Omron CX-Programmer project NewProject (CX-Programmer 9.75)

# PLC NewPLC1: CP2E-N N

## Global symbols (name address type ; comment)
0.00 BOOL  ; PB Start M1
0.01 BOOL  ; PB Stop M1
0.02 BOOL  ; SS FWD M1
0.03 BOOL  ; SS RVS M1
0.04 BOOL  ; Emergency Stop
0.05 BOOL  ; Sensor M1
0.06 BOOL  ; Trip CNT M1
100.00 BOOL  ; Trip M1
100.01 BOOL  ; Contactor M1
100.02 BOOL  ; Relay FWD M1
100.03 BOOL  ; Relay RVS M1
101.00 BOOL  ; Trip M2
101.01 BOOL  ; Contactor M2
101.02 BOOL  ; Relay FWD M2
101.03 BOOL  ; Relay RVS M2
170.01 BOOL  ; LOCK START FWD VER
1.00 BOOL  ; PB Start M2
1.01 BOOL  ; PB Stop M2
1.02 BOOL  ; SS FWD M2
1.03 BOOL  ; SS RVS M2
1.04 BOOL  ; Sensor M2
1.05 BOOL  ; Trip CNT M2
21.00 BOOL  ; ls vertical fwd
21.01 BOOL  ; ls vertical rev
21.02 BOOL  ; ls horizontal fwd
21.03 BOOL  ; ls horizontal rev
60.00 BOOL  ; M1_achieved'
70.01 BOOL  ; LOCK START FWD HOR
70.02 BOOL  ; LOCK START REV HOR
C000 BOOL  ; Siklus M1
C001 BOOL  ; Siklus M2
C002 BOOL  ; Siklus M1
C003 BOOL  ; Siklus M2
C010 BOOL  ; Siklus (1) M1
C011 BOOL  ; Siklus (2) M1
C110 BOOL  ; Siklus (1) M2
C111 BOOL  ; Siklus (2) M2
D0 CHANNEL  ; Input Siklus M1
D10 CHANNEL  ; Input Siklus M2
D100 CHANNEL  ; '
D20 CHANNEL  ; Input Siklus M1
D30 CHANNEL  ; Input Siklus M2
D5400 CHANNEL  ; Counter_test
D5410 CHANNEL  ; Counter_target
D600 CHANNEL  ; Input Siklus M1
D660 CHANNEL  ; Input Siklus M2
W0.00 BOOL  ; H.PB Start M1
W0.01 BOOL  ; H.PB Stop M1
W0.02 BOOL  ; H.SS FWD M1
W0.03 BOOL  ; H.SS RVS M1
W0.04 BOOL  ; H.Emergency Stop
W0.05 BOOL  ; H.Sensor M1
W0.06 BOOL  ; H.Trip CNT M1
W0.07 BOOL  ; LS Left M1
W0.08 BOOL  ; LS Right M1
W100.00 BOOL  ; H.Trip M1
W100.01 BOOL  ; H.CONTACTOR M1
W100.02 BOOL  ; H.Relay FWD M1
W100.03 BOOL  ; H.Relay RVS M1
W101.00 BOOL  ; H.Trip M2
W101.01 BOOL  ; H.CONTACTOR M2
W101.02 BOOL  ; H.Relay FWD M2
W101.03 BOOL  ; H.Relay RVS M2
W1.00 BOOL  ; H.PB Start M2
W1.01 BOOL  ; H.PB Stop M2
W1.02 BOOL  ; H.SS FWD M2
W1.03 BOOL  ; H.SS RVS M2
W1.04 BOOL  ; H.Sensor M2
W1.05 BOOL  ; H.Trip CNT M2
W1.06 BOOL  ; LS Left M2
W1.07 BOOL  ; LS Right M2
W20.01 BOOL  ; CYCLE 50 RB
W20.02 BOOL  ; CYCLE 100 RB
W20.03 BOOL  ; Mix M1
W20.04 BOOL  ; Mix M2
W21.02 BOOL  ; Cycle 100rb mix
W2.00 BOOL  ; Reset M1
W2.02 BOOL  ; Reset M2
W60.01 BOOL  ; W CNT 1
W61.01 BOOL  ; W CNT 2

## Program NewProgram1 (cyclic task 0)
Local symbols
CO UINT_BCD
D100D20 INT
DD5400 UDINT
P_0_01s BOOL
P_off BOOL
p_0_1s BOOL
p_off BOOL

### Section Alat_Uji_Pedal
; PUSH BUTTON

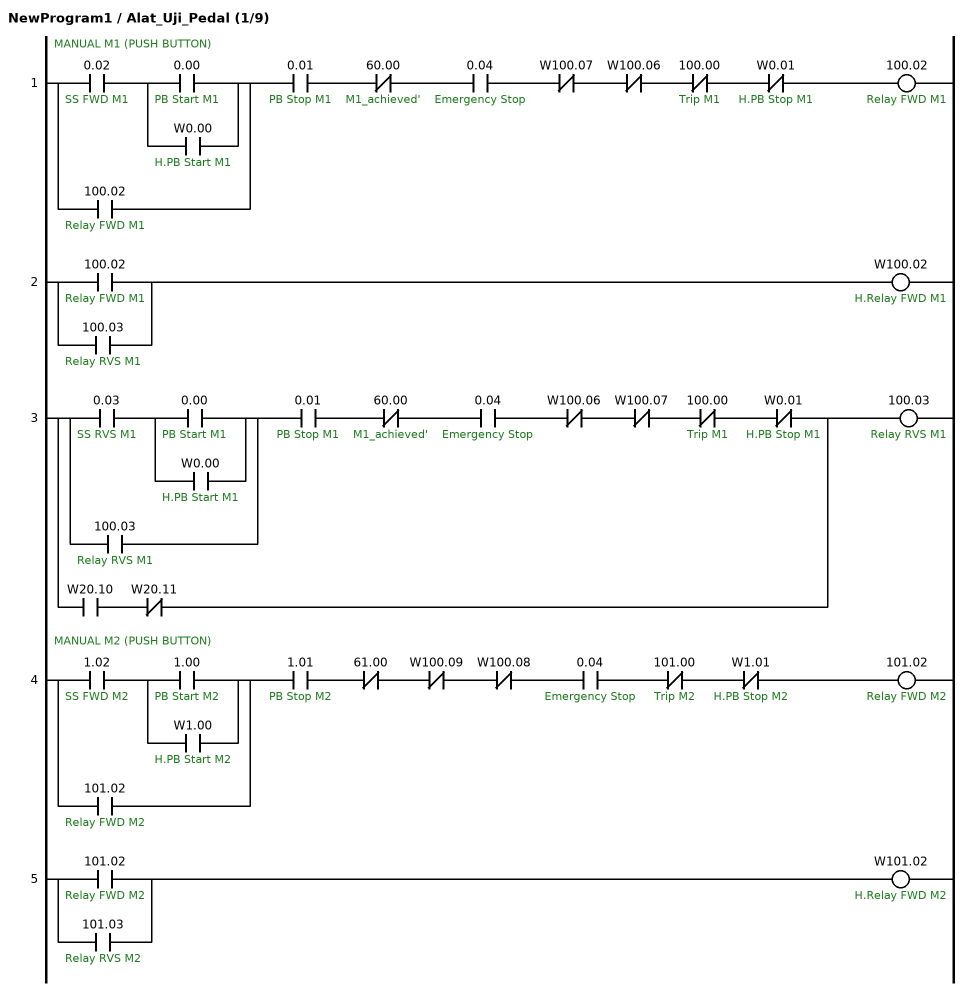
; rung 1: MANUAL M1 (PUSH BUTTON)
LD 0.02  ; SS FWD M1
LD 0.00  ; PB Start M1
OR W0.00  ; H.PB Start M1
ANDLD
OR 100.02  ; Relay FWD M1
AND 0.01  ; PB Stop M1
ANDNOT 60.00  ; M1_achieved'
AND 0.04  ; Emergency Stop
ANDNOT W100.07
ANDNOT W100.06
ANDNOT 100.00  ; Trip M1
ANDNOT W0.01  ; H.PB Stop M1
OUT 100.02  ; Relay FWD M1
; rung 2
LD 100.02  ; Relay FWD M1
OR 100.03  ; Relay RVS M1
OUT W100.02  ; H.Relay FWD M1
; rung 3
LD 0.03  ; SS RVS M1
LD 0.00  ; PB Start M1
OR W0.00  ; H.PB Start M1
ANDLD
OR 100.03  ; Relay RVS M1
AND 0.01  ; PB Stop M1
ANDNOT 60.00  ; M1_achieved'
AND 0.04  ; Emergency Stop
ANDNOT W100.06
ANDNOT W100.07
ANDNOT 100.00  ; Trip M1
ANDNOT W0.01  ; H.PB Stop M1
LD W20.10
ANDNOT W20.11
ORLD
OUT 100.03  ; Relay RVS M1
; rung 4: MANUAL M2 (PUSH BUTTON)
LD 1.02  ; SS FWD M2
LD 1.00  ; PB Start M2
OR W1.00  ; H.PB Start M2
ANDLD
OR 101.02  ; Relay FWD M2
AND 1.01  ; PB Stop M2
ANDNOT 61.00
ANDNOT W100.09
ANDNOT W100.08
AND 0.04  ; Emergency Stop
ANDNOT 101.00  ; Trip M2
ANDNOT W1.01  ; H.PB Stop M2
OUT 101.02  ; Relay FWD M2
; rung 5
LD 101.02  ; Relay FWD M2
OR 101.03  ; Relay RVS M2
OUT W101.02  ; H.Relay FWD M2

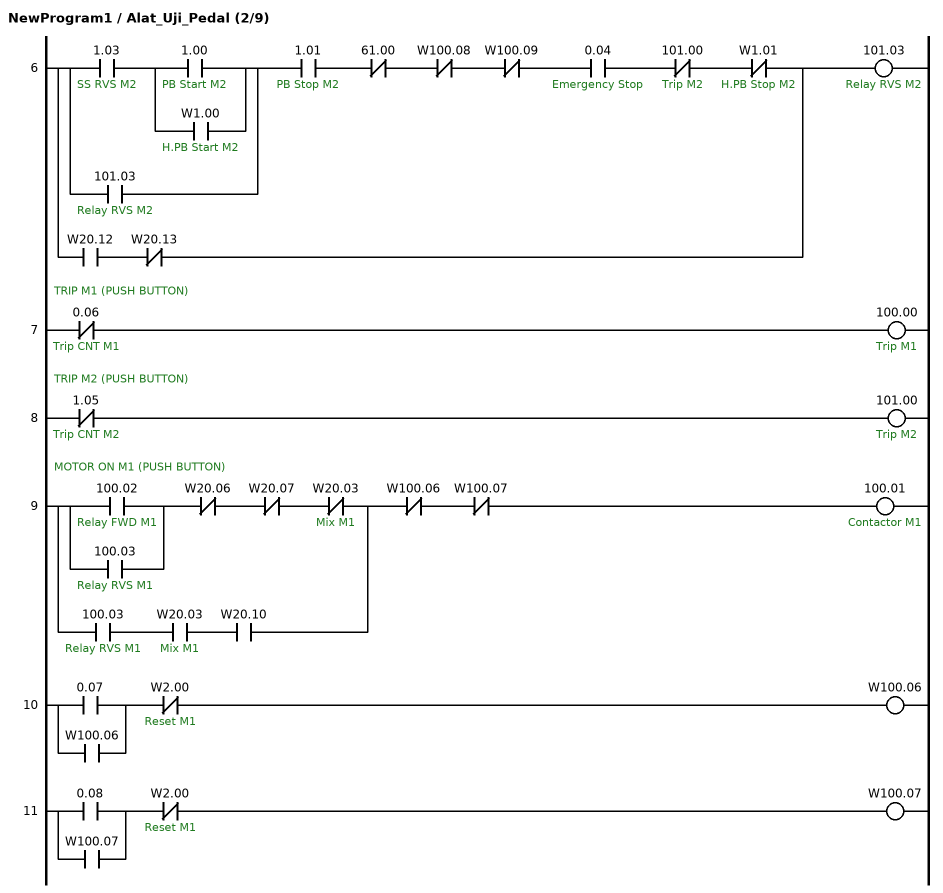
; rung 6
LD 1.03  ; SS RVS M2
LD 1.00  ; PB Start M2
OR W1.00  ; H.PB Start M2
ANDLD
OR 101.03  ; Relay RVS M2
AND 1.01  ; PB Stop M2
ANDNOT 61.00
ANDNOT W100.08
ANDNOT W100.09
AND 0.04  ; Emergency Stop
ANDNOT 101.00  ; Trip M2
ANDNOT W1.01  ; H.PB Stop M2
LD W20.12
ANDNOT W20.13
ORLD
OUT 101.03  ; Relay RVS M2
; rung 7: TRIP M1 (PUSH BUTTON)
LDNOT 0.06  ; Trip CNT M1
OUT 100.00  ; Trip M1
; rung 8: TRIP M2 (PUSH BUTTON)
LDNOT 1.05  ; Trip CNT M2
OUT 101.00  ; Trip M2
; rung 9: MOTOR ON M1 (PUSH BUTTON)
LD 100.02  ; Relay FWD M1
OR 100.03  ; Relay RVS M1
ANDNOT W20.06
ANDNOT W20.07
ANDNOT W20.03  ; Mix M1
LD 100.03  ; Relay RVS M1
AND W20.03  ; Mix M1
AND W20.10
ORLD
ANDNOT W100.06
ANDNOT W100.07
OUT 100.01  ; Contactor M1
; rung 10
LD 0.07
OR W100.06
ANDNOT W2.00  ; Reset M1
OUT W100.06
; rung 11
LD 0.08
OR W100.07
ANDNOT W2.00  ; Reset M1
OUT W100.07

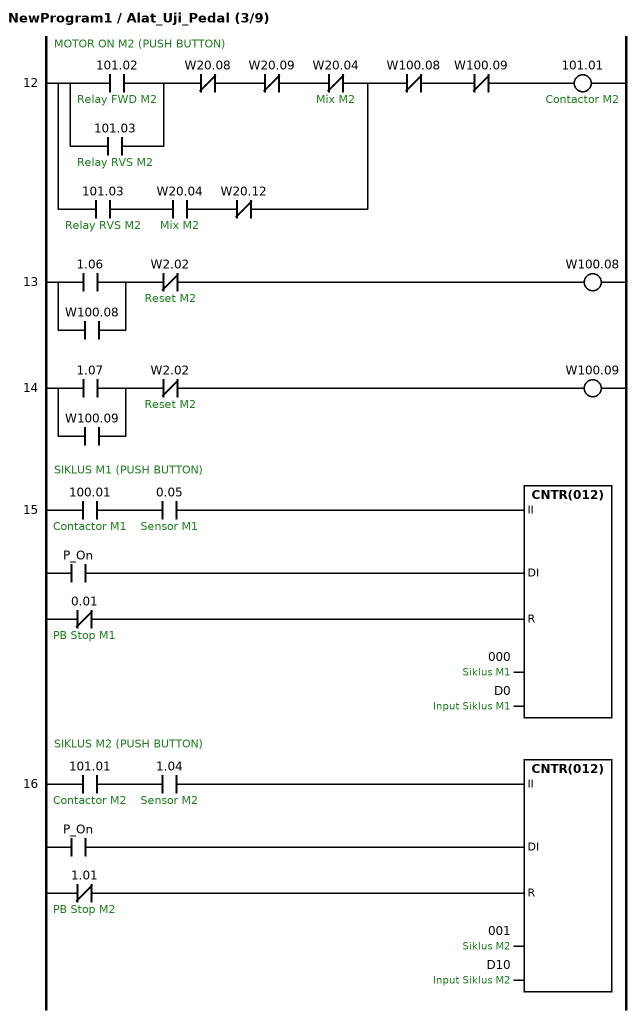
; rung 12: MOTOR ON M2 (PUSH BUTTON)
LD 101.02  ; Relay FWD M2
OR 101.03  ; Relay RVS M2
ANDNOT W20.08
ANDNOT W20.09
ANDNOT W20.04  ; Mix M2
LD 101.03  ; Relay RVS M2
AND W20.04  ; Mix M2
ANDNOT W20.12
ORLD
ANDNOT W100.08
ANDNOT W100.09
OUT 101.01  ; Contactor M2
; rung 13
LD 1.06
OR W100.08
ANDNOT W2.02  ; Reset M2
OUT W100.08
; rung 14
LD 1.07
OR W100.09
ANDNOT W2.02  ; Reset M2
OUT W100.09
; rung 15: SIKLUS M1 (PUSH BUTTON)
LD 100.01  ; Contactor M1
AND 0.05  ; Sensor M1
LD P_On
LDNOT 0.01  ; PB Stop M1
CNTR(012) 000 D0  ; Input Siklus M1, Siklus M1
; rung 16: SIKLUS M2 (PUSH BUTTON)
LD 101.01  ; Contactor M2
AND 1.04  ; Sensor M2
LD P_On
LDNOT 1.01  ; PB Stop M2
CNTR(012) 001 D10  ; Input Siklus M2, Siklus M2

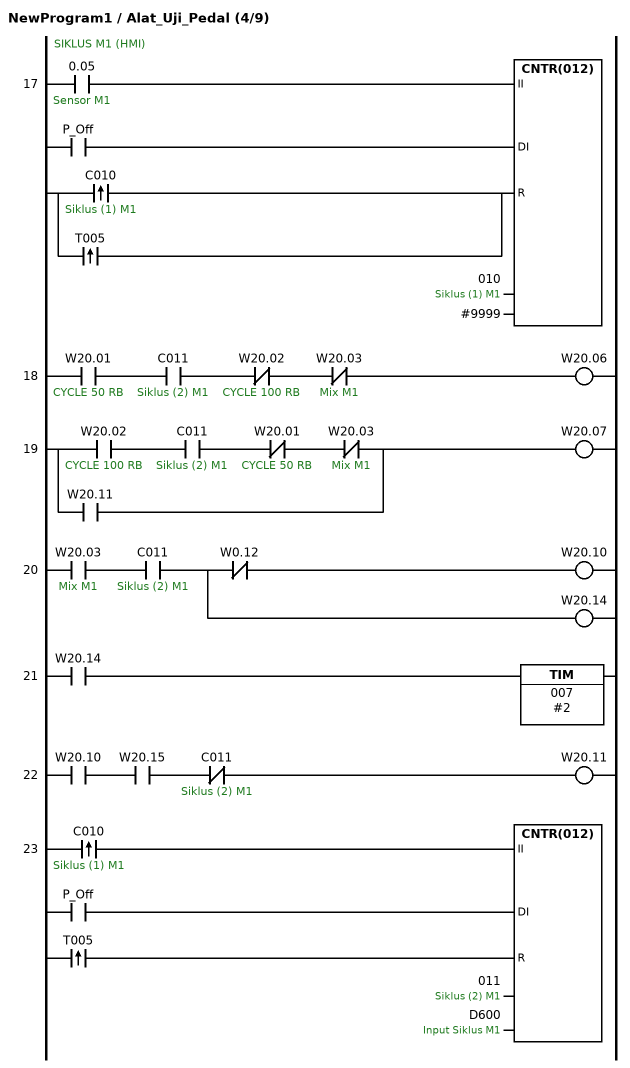
; rung 17: SIKLUS M1 (HMI)
LD 0.05  ; Sensor M1
LD P_Off
@LD C010  ; Siklus (1) M1
@OR T005
CNTR(012) 010 #9999  ; Siklus (1) M1
; rung 18
LD W20.01  ; CYCLE 50 RB
AND C011  ; Siklus (2) M1
ANDNOT W20.02  ; CYCLE 100 RB
ANDNOT W20.03  ; Mix M1
OUT W20.06
; rung 19
LD W20.02  ; CYCLE 100 RB
AND C011  ; Siklus (2) M1
ANDNOT W20.01  ; CYCLE 50 RB
ANDNOT W20.03  ; Mix M1
OR W20.11
OUT W20.07
; rung 20
LD W20.03  ; Mix M1
AND C011  ; Siklus (2) M1
OUT TR0
ANDNOT W0.12
OUT W20.10
LD TR0
OUT W20.14
; rung 21
LD W20.14
TIM 007 #2
; rung 22
LD W20.10
AND W20.15
ANDNOT C011  ; Siklus (2) M1
OUT W20.11
; rung 23
@LD C010  ; Siklus (1) M1
LD P_Off
@LD T005
CNTR(012) 011 D600  ; Input Siklus M1, Siklus (2) M1

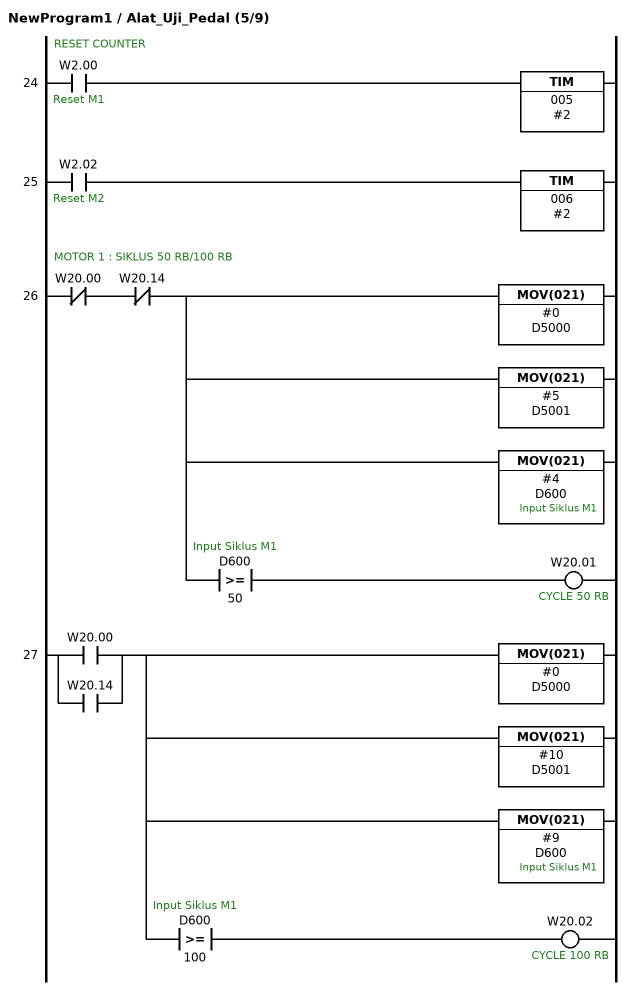
; rung 24: RESET COUNTER
LD W2.00  ; Reset M1
TIM 005 #2
; rung 25
LD W2.02  ; Reset M2
TIM 006 #2
; rung 26: MOTOR 1 : SIKLUS 50 RB/100 RB
LDNOT W20.00
ANDNOT W20.14
MOV(021) #0 D5000
MOV(021) #5 D5001
MOV(021) #4 D600  ; Input Siklus M1
AND>=(325) D600 50  ; Input Siklus M1
OUT W20.01  ; CYCLE 50 RB
; rung 27
LD W20.00
OR W20.14
MOV(021) #0 D5000
MOV(021) #10 D5001
MOV(021) #9 D600  ; Input Siklus M1
AND>=(325) D600 100  ; Input Siklus M1
OUT W20.02  ; CYCLE 100 RB

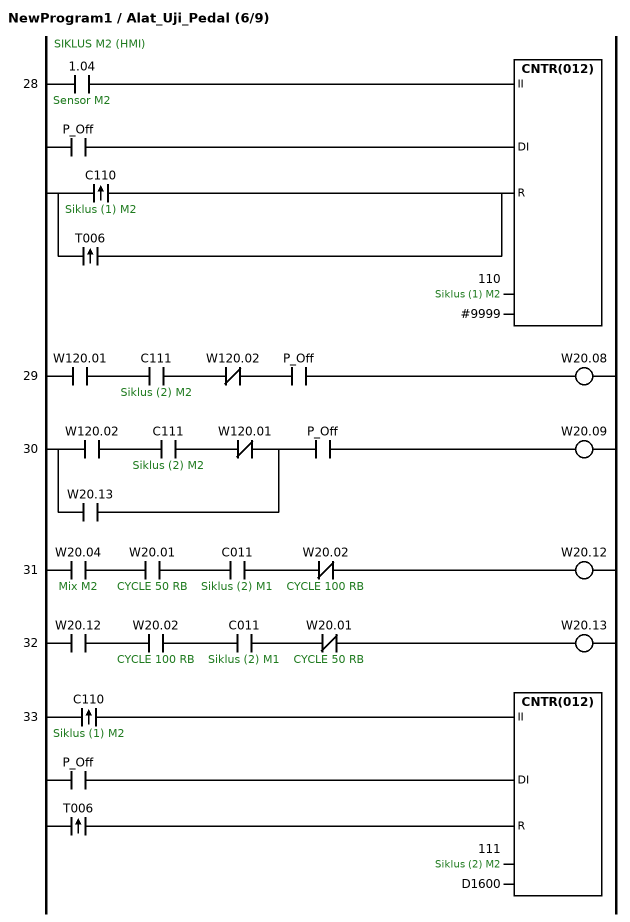
; rung 28: SIKLUS M2 (HMI)
LD 1.04  ; Sensor M2
LD P_Off
@LD C110  ; Siklus (1) M2
@OR T006
CNTR(012) 110 #9999  ; Siklus (1) M2
; rung 29
LD W120.01
AND C111  ; Siklus (2) M2
ANDNOT W120.02
AND P_Off
OUT W20.08
; rung 30
LD W120.02
AND C111  ; Siklus (2) M2
ANDNOT W120.01
OR W20.13
AND P_Off
OUT W20.09
; rung 31
LD W20.04  ; Mix M2
AND W20.01  ; CYCLE 50 RB
AND C011  ; Siklus (2) M1
ANDNOT W20.02  ; CYCLE 100 RB
OUT W20.12
; rung 32
LD W20.12
AND W20.02  ; CYCLE 100 RB
AND C011  ; Siklus (2) M1
ANDNOT W20.01  ; CYCLE 50 RB
OUT W20.13
; rung 33
@LD C110  ; Siklus (1) M2
LD P_Off
@LD T006
CNTR(012) 111 D1600  ; Siklus (2) M2

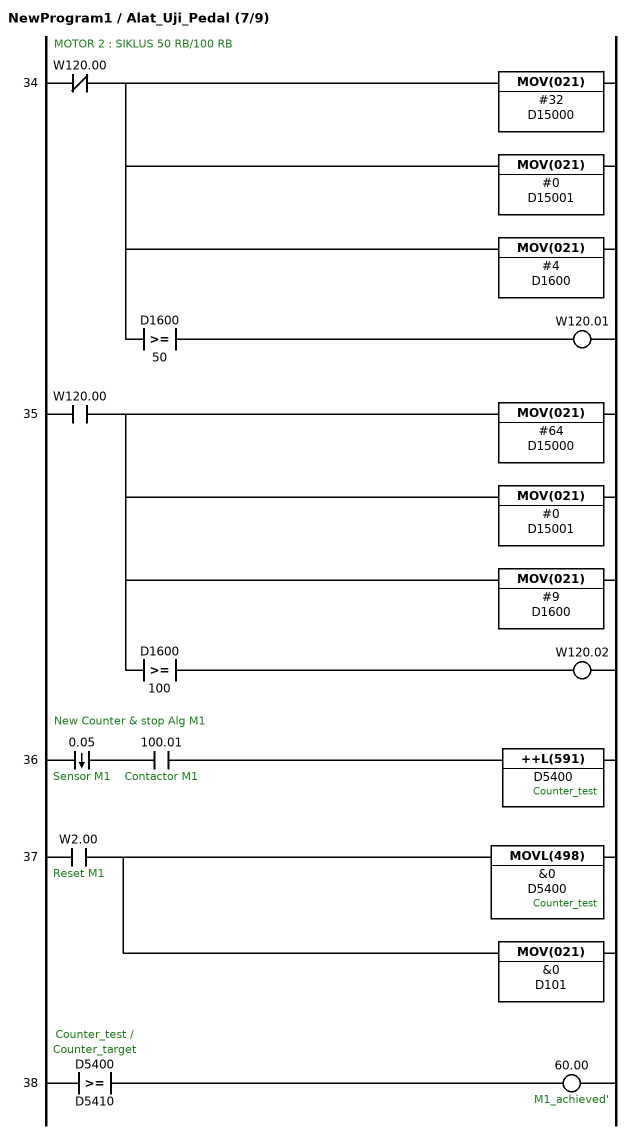
; rung 34: MOTOR 2 : SIKLUS 50 RB/100 RB
LDNOT W120.00
MOV(021) #32 D15000
MOV(021) #0 D15001
MOV(021) #4 D1600
AND>=(325) D1600 50
OUT W120.01
; rung 35
LD W120.00
MOV(021) #64 D15000
MOV(021) #0 D15001
MOV(021) #9 D1600
AND>=(325) D1600 100
OUT W120.02
; rung 36: New Counter & stop Alg M1
%LD 0.05  ; Sensor M1
AND 100.01  ; Contactor M1
++L(591) D5400  ; Counter_test
; rung 37
LD W2.00  ; Reset M1
MOVL(498) &0 D5400  ; Counter_test
MOV(021) &0 D101
; rung 38
LD>=L(326) D5400 D5410  ; Counter_test, Counter_target
OUT 60.00  ; M1_achieved'

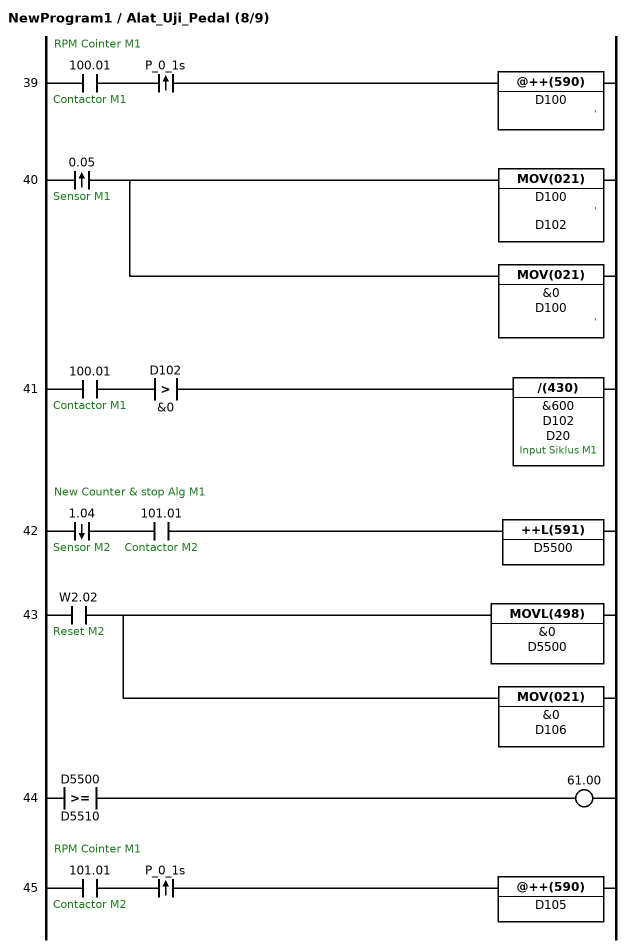
; rung 39: RPM Cointer M1
LD 100.01  ; Contactor M1
@AND P_0_1s
@++(590) D100  ; '
; rung 40
@LD 0.05  ; Sensor M1
MOV(021) D100 D102  ; '
MOV(021) &0 D100  ; '
; rung 41
LD 100.01  ; Contactor M1
AND>(320) D102 &0
/(430) &600 D102 D20  ; Input Siklus M1
; rung 42: New Counter & stop Alg M1
%LD 1.04  ; Sensor M2
AND 101.01  ; Contactor M2
++L(591) D5500
; rung 43
LD W2.02  ; Reset M2
MOVL(498) &0 D5500
MOV(021) &0 D106
; rung 44
LD>=L(326) D5500 D5510
OUT 61.00
; rung 45: RPM Cointer M1
LD 101.01  ; Contactor M2
@AND P_0_1s
@++(590) D105

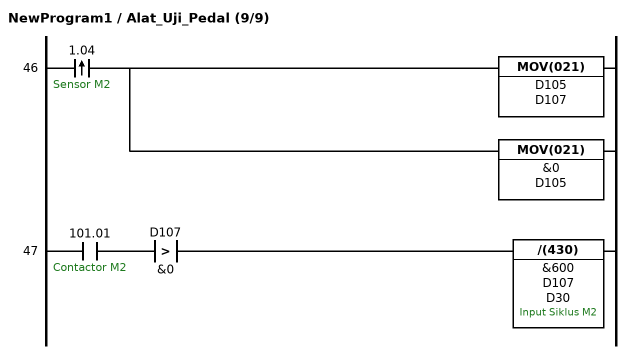
; rung 46
@LD 1.04  ; Sensor M2
MOV(021) D105 D107
MOV(021) &0 D105
; rung 47
LD 101.01  ; Contactor M2
AND>(320) D107 &0
/(430) &600 D107 D30  ; Input Siklus M2

### Section END
; rung 0
END(001)